(* PLC project Unnamed, Unknown Unnamed 1 *)
(* stored: creationDateTime 2024-09-16T10:11:28, modificationDateTime 2024-09-16T10:28:46 *)

PROGRAM water_tank

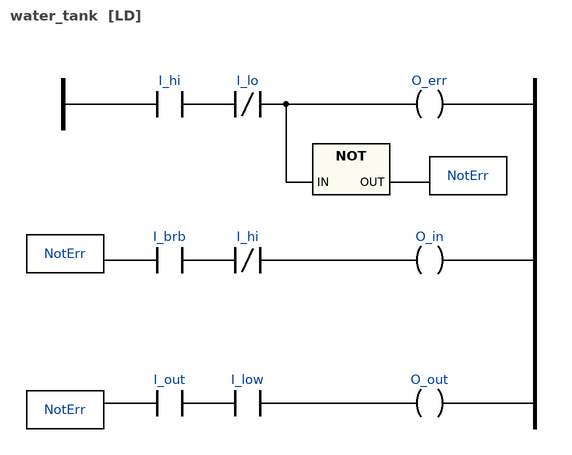
(* LD diagram, written out as Structured Text *)
O_err := I_hi AND NOT I_lo;
NotErr := NOT (I_hi AND NOT I_lo);
O_in := NotErr AND I_brb AND NOT I_hi;
O_out := NotErr AND I_out AND I_low;
END_PROGRAM

CONFIGURATION Config0
  RESOURCE Res0 ON PLC
    TASK task0(INTERVAL := T#20ms, PRIORITY := 0);
    PROGRAM instance0 WITH task0 : water_tank;
  END_RESOURCE
END_CONFIGURATION
